TEXTLIST ModoDescripcion
  0 = 'Parada en el estado inicial'
  1 = 'Parada a final de ciclo'
  2 = 'Parada pedida'
  3 = 'Parada obtenida'
  4 = 'Recuperación del defecto'
  5 = 'Puesta en el estado inicial'
  6 = 'Puesta en un estado determinado'
  7 = 'Produccion normal'
  8 = 'Marchas de preparación'
  9 = 'Marchas de cierre'
  10 = 'M. verificacion en desorden'
  11 = 'M. verificacion en orden'
  12 = 'Marchas de prueba'
  13 = 'Emergencia'
  14 = 'Tratamiento de los defectos'
  15 = 'Producción con defectos'
   = ''
END_TEXTLIST

(* stored: Version 1.1.0.1, ProductVersion 3.1.4024.12
   TextList ModoDescripcion: Id {11f39ec0-46ce-4d0f-b0ba-275a3ffeb426} *)
